Fanuc KAREL source: KT00543.KL

PROGRAM KT00543
%NOLOCKGROUP
VAR
  P1: JOINTPOS
  P2: XYZWPREXT
  OUT: BOOLEAN
BEGIN
    P2.Y = 2.0
  OUT = P1 >=< P2
END KT00543
